DATA_BLOCK "Simulation_DB"
{ S7_Optimized_Access := 'TRUE' }
"Simulation"


BEGIN

END_DATA_BLOCK
